// TIA Portal V20 export
TYPE "LKinCtrl_typeRelShift"
   STRUCT
      coordinates : Array[1..6] of LReal;   // Coordinates of relative CS shift
      coordinateSystem : DInt;   // Base coordinate system which shift is applied
      shiftActive : Bool;   // TRUE: Shift is active
   END_STRUCT;
END_TYPE
